# EPICS StreamDevice protocol: E2010App/Db/ZIROXE2010.proto
#ZIROX ELECTRONIC E2010

Terminator = CR;

readoxygen {out "M2"; in "M2%f ";}
readvoltage {out "A1"; in "A1%f ";}
readtemp {out "A2"; in "A2%f ";}
